Staubli VAL3: AXIS7.pjx

--- AXIS7.pjx ---
Parameters version=s7.2.1 stackSize=5000 millimeterUnit=true
Program file=del.pgx
Program file=find.pgx
Program file=findValue.pgx
Program file=get.pgx
Program file=getSize.pgx
Program file=getType.pgx
Program file=getValue.pgx
Program file=getVelocity.pgx
Program file=loadCycle.pgx
Program file=new.pgx
Program file=onEdit.pgx
Program file=onInsert.pgx
Program file=onProgEnd.pgx
Program file=onRun.pgx
Program file=onStart.pgx
Program file=onStop.pgx
Program file=set.pgx
Program file=setValue.pgx
Program file=setVelocity.pgx
Data file=AXIS7.dtx
Library alias=language path=Disk://kernel/language/language.pjx
Library alias=use path=Disk://kernel/userPage/userPage.pjx

--- AXIS7.dtx ---
public aio MbAI_a8Axispose = {link=ModbusSrv-0\Modbus-Word\MbAI_a8Axispose}
public aio MbAI_aCurPosH = {link=ModbusSrv-0\Modbus-Word\MbAI_aCurPosH}
public aio MbAI_aCurPosL = {link=ModbusSrv-0\Modbus-Word\MbAI_aCurPosL}
public aio MbAI_aUnused4 = {link=ModbusSrv-0\Modbus-Word\MbAI_aUnused4}
public aio MbAI_b8MotorErr = {link=ModbusSrv-0\Modbus-Word\MbAI_b8MotorError}
public aio MbAI_b8MotorPow = {link=ModbusSrv-0\Modbus-Word\MbAI_b8MotorPower}
public aio MbAI_bAxis7Reac = {link=ModbusSrv-0\Modbus-Word\MbAI_bAxis7Reached}
public aio MbAI_bAxis8Reac = {link=ModbusSrv-0\Modbus-Word\MbAI_bAxis8Reached}
public aio MbAI_bBackHome = {link=ModbusSrv-0\Modbus-Word\MbAI_bBackHome}
public aio MbAI_bDownLimit = {link=ModbusSrv-0\Modbus-Word\MbAI_bDownLimit}
public aio MbAI_bEndCycl = {link=ModbusSrv-0\Modbus-Word\MbAI_bEndCycl}
public aio MbAI_bHomeDone = {link=ModbusSrv-0\Modbus-Word\MbAI_bHomeDone}
public aio MbAI_bHomeLimit = {link=ModbusSrv-0\Modbus-Word\MbAI_bHomeLimit}
public aio MbAI_bIsHome = {link=ModbusSrv-0\Modbus-Word\MbAI_bIsHome}
public aio MbAI_bMotorErro = {link=ModbusSrv-0\Modbus-Word\MbAI_bMotorError}
public aio MbAI_bMotorPowe = {link=ModbusSrv-0\Modbus-Word\MbAI_bMotorPower}
public aio MbAI_bOutAlarm = {link=ModbusSrv-0\Modbus-Word\MbAI_bOutAlarm}
public aio MbAI_bPowerOn = {link=ModbusSrv-0\Modbus-Word\MbAI_bPowerOn}
public aio MbAI_bStartCycl = {link=ModbusSrv-0\Modbus-Word\MbAI_bStartCycl}
public aio MbAI_bUnused1 = {link=ModbusSrv-0\Modbus-Word\MbAI_bUnused1}
public aio MbAI_bUnused10 = {link=ModbusSrv-0\Modbus-Word\MbAI_bUnused10}
public aio MbAI_bUnused11 = {link=ModbusSrv-0\Modbus-Word\MbAI_bUnused11}
public aio MbAI_bUnused2 = {link=ModbusSrv-0\Modbus-Word\MbAI_bUnused2}
public aio MbAI_bUnused3 = {link=ModbusSrv-0\Modbus-Word\MbAI_bUnused3}
public aio MbAI_bUnused5 = {link=ModbusSrv-0\Modbus-Word\MbAI_bUnused5}
public aio MbAI_bUnused6 = {link=ModbusSrv-0\Modbus-Word\MbAI_bUnused6}
public aio MbAI_bUnused7 = {link=ModbusSrv-0\Modbus-Word\MbAI_bUnused7}
public aio MbAI_bUnused8 = {link=ModbusSrv-0\Modbus-Word\MbAI_bUnused8}
public aio MbAI_bUnused9 = {link=ModbusSrv-0\Modbus-Word\MbAI_bUnused9}
public aio MbAI_bUpLimit = {link=ModbusSrv-0\Modbus-Word\MbAI_bUpLimit}
public aio MbAO_aAxis7Puls = {link=ModbusSrv-0\Modbus-Word\MbAO_aAxis7Pulse}
public aio MbAO_aAxis8Puls = {link=ModbusSrv-0\Modbus-Word\MbAO_aAxis8Pulse}
public aio MbAO_aJogVelo = {link=ModbusSrv-0\Modbus-Word\MbAO_aJogVelo}
public aio MbAO_aJogVelo8 = {link=ModbusSrv-0\Modbus-Word\MbAO_aJogVelo8}
public aio MbAO_aMoveDis = {link=ModbusSrv-0\Modbus-Word\MbAO_aMoveDis}
public aio MbAO_aMoveDis8 = {link=ModbusSrv-0\Modbus-Word\MbAO_aMoveDis8}
public aio MbAO_aMovePosH = {link=ModbusSrv-0\Modbus-Word\MbAO_aMovePosH}
public aio MbAO_aMovePosH8 = {link=ModbusSrv-0\Modbus-Word\MbAO_aMovePosH8}
public aio MbAO_aMovePosL = {link=ModbusSrv-0\Modbus-Word\MbAO_aMovePosL}
public aio MbAO_aMovePosL8 = {link=ModbusSrv-0\Modbus-Word\MbAO_aMovePosL8}
public aio MbAO_aUnused10 = {link=ModbusSrv-0\Modbus-Word\MbAO_aUnused10}
public aio MbAO_aUnused11 = {link=ModbusSrv-0\Modbus-Word\MbAO_aUnused11}
public aio MbAO_aUnused6 = {link=ModbusSrv-0\Modbus-Word\MbAO_aUnused6}
public aio MbAO_aUnused7 = {link=ModbusSrv-0\Modbus-Word\MbAO_aUnused7}
public aio MbAO_aUnused8 = {link=ModbusSrv-0\Modbus-Word\MbAO_aUnused8}
public aio MbAO_aUnused9 = {link=ModbusSrv-0\Modbus-Word\MbAO_aUnused9}
public aio MbAO_aVelocity = {link=ModbusSrv-0\Modbus-Word\MbAO_aVelocity}
public aio MbAO_aVelocity8 = {link=ModbusSrv-0\Modbus-Word\MbAO_aVelocity8}
public aio MbAO_b7Axis = {link=ModbusSrv-0\Modbus-Word\MbAO_b7Axis}
public aio MbAO_b8Axis = {link=ModbusSrv-0\Modbus-Word\MbAO_b8Axis}
public aio MbAO_bAxis7Dire = {link=ModbusSrv-0\Modbus-Word\MbAO_bAxis7Direction}
public aio MbAO_bAxis7Home = {link=ModbusSrv-0\Modbus-Word\MbAO_bAxis7Home}
public aio MbAO_bAxis8Dire = {link=ModbusSrv-0\Modbus-Word\MbAO_bAxis8Direction}
public aio MbAO_bMoveDir = {link=ModbusSrv-0\Modbus-Word\MbAO_bMoveDir}
public aio MbAO_bMoveDirM = {link=ModbusSrv-0\Modbus-Word\MbAO_bMoveDirM}
public aio MbAO_bMovePos8 = {link=ModbusSrv-0\Modbus-Word\MbAO_bMovePos8}
public aio MbAO_bMoveToPos = {link=ModbusSrv-0\Modbus-Word\MbAO_bMoveToPos}
public aio MbAO_bRecordPos = {link=ModbusSrv-0\Modbus-Word\MbAO_bRecordPos}
public aio MbAO_bResetErr = {link=ModbusSrv-0\Modbus-Word\MbAO_bResetErr}
public aio MbAO_bStopMotor = {link=ModbusSrv-0\Modbus-Word\MbAO_bStopMotor}
public aio MbAO_bUnused1 = {link=ModbusSrv-0\Modbus-Word\MbAO_bUnused1}
public aio MbAO_bUnused2 = {link=ModbusSrv-0\Modbus-Word\MbAO_bUnused2}
public aio MbAO_bUnused3 = {link=ModbusSrv-0\Modbus-Word\MbAO_bUnused3}
public aio MbAO_bUnused4 = {link=ModbusSrv-0\Modbus-Word\MbAO_bUnused4}
public aio MbAO_bUnused5 = {link=ModbusSrv-0\Modbus-Word\MbAO_bUnused5}
public bool bAxisRun
num i = 6
public num nSaveaxis[7]
  [0] = 17569
  [1] = 17753
  [2] = 17775
  [3] = 17555
  [4] = 17803
  [5] = 17805
  [6] = 17722
public num nSaveaxis1[7]
  [0] = 36925
  [1] = 31321
  [2] = 60066
  [3] = 25553
  [4] = 27683
  [5] = 48927
  [6] = 32566
public num nVelocity[7]
  [0] = 8
  [1] = 8
  [2] = 8
  [3] = 8
  [4] = 8
  [5] = 8
  [6] = 8
string l_sItem = "PStart"
public string sItems
public string sSaveaxis[7]
  [0] = "workPos"
  [1] = "p1"
  [2] = "PStart"
  [3] = "P_001"
  [4] = "P_002"
  [5] = "PEnd"
  [6] = "PSychro"

--- del.pgx ---
public program del(num x_nIndex)
begin
  //delete(saveAxis[x_nIndex])
  if size(nSaveaxis)>1
    $ddel(nSaveaxis,x_nIndex)
    $ddel(nSaveaxis1,x_nIndex)
    $ddel(sSaveaxis,x_nIndex)
    $ddel(nVelocity,x_nIndex)
  endIf
end

--- find.pgx ---
public program find(string& x_sItem[], bool& x_bFound[])
begin
  //
  // find one item in the list
  //
  for i=0 to size(sSaveaxis)-1
    if sSaveaxis[i]==x_sItem
      x_bFound=true
      return
    endIf
  endFor
end

--- get.pgx ---
public program get(string& x_sItem[], num x_nIndex)
begin
  //
  // get one element from the list
  //
  x_sItem=sSaveaxis[x_nIndex]
end

--- getSize.pgx ---
public program getSize(num& x_nSize[])
begin
  //
  // get the size of the list
  //
  x_nSize=size(sSaveaxis)
end

--- getValue.pgx ---
public program getValue(num& x_nValue[], num& x_nIndex[], num& x_nValue1[])
begin
  //
  // get the size of the list
  //
  x_nValue=nSaveaxis[x_nIndex]
  //x_nValue=nVelocity[x_nIndex]
  x_nValue1=nSaveaxis1[x_nIndex]
end

--- getVelocity.pgx ---
public program getVelocity(string& x_sItem[], num& x_nVelocity[])
  local num l_nSize
begin
  call getSize(l_nSize)
  for i=0 to l_nSize
    call get(l_sItem,i)
    if l_sItem==x_sItem
      x_nVelocity=nVelocity[i]
      return
      //go back
    endIf
  endFor
end

--- new.pgx ---
public program new(string x_sItem, num x_nIndex)
begin
  // insert a new item
  //insert(saveAxis[x_nIndex])
  $dins(nSaveaxis,size(nSaveaxis))
  $dins(nSaveaxis1,size(nSaveaxis1))
  $dins(sSaveaxis,size(sSaveaxis))
  $dins(nVelocity,size(nVelocity))
  sSaveaxis[size(sSaveaxis)-1]=x_sItem
  nVelocity[size(nVelocity)-1]=8
  ? x_sItem
end

--- onInsert.pgx ---
public program onInsert(string& x_sItem[])
  local string l_sItem
  local string l_sEvent
  local num l_nSize
  local num l_nKey
begin
  //
  // compose the string
  // call getType(l_sItem)
  // x_sItem=l_sItem+" ???"
  //
  // insert all the saveAxis value from the list
  cls()
  call language:message(l_sEvent,65)
  call use:clear(0,13)
  call use:typeCenter(13,l_sEvent,40,true)
  x_sItem=""
  call use:setSizeList(19,0,19,10)
  call use:listcreate("AXIS7")
  l_nSize=size(nSaveaxis)
  for i=0 to l_nSize-1
    l_sEvent=sSaveaxis[i]
    call use:listadd(l_sEvent)
  endFor
  call use:listupdate(0)
  do
    l_nKey=getKey()
    call use:listevent(l_nKey,i,l_sEvent)
    delay(0)
  until l_nKey==255 or l_nKey==270
  if l_nKey==270
    x_sItem="AXIS7>"+l_sEvent
  endIf
  call use:nullKey(l_nKey)
  delay(0)
end

--- onProgEnd.pgx ---
public program onProgEnd(string& x_sItem[])
begin
  //
  // Done, when one program has finished
  //
end

--- onRun.pgx ---
public program onRun(string& x_sItem[])
  local num l_nValue
  local num l_nValue1
  local num l_nVelocity
begin
  //
  // Done, when you execute it
  //
  ////  call findValue(x_sItem,l_nValue)
  ////  aioSet(io:movePulse,l_nValue)
  ////  io:move=true
  ////  delay(0.5)
  ////  io:move=false
  ////  wait(io:atPosition==true or isKeyPressed(255))
  if aioGet(MbAI_bBackHome)!=1
    popUpMsg("7轴未回零位，请先执行回零位操作")
    return
  endIf
  aioSet(MbAO_b7Axis,1)
  aioSet(MbAO_aMoveDis,0)
  aioSet(MbAO_bMoveToPos,0)
  bAxisRun=true
//  aioSet(MbAI_bAxis7Reac,0)
  delay(0.5)
  call findValue(x_sItem,l_nValue,l_nValue1)
  call getVelocity(x_sItem,l_nVelocity)
  l_nVelocity=l_nVelocity*1000/60
  aioSet(MbAO_aMovePosL,l_nValue)
  aioSet(MbAO_aMovePosH,l_nValue1)
  aioSet(MbAO_aVelocity,l_nVelocity)
  aioSet(MbAO_bMoveToPos,1)
  delay(0.5)
  wait(aioGet(MbAI_bAxis7Reac)==0)
  wait(aioGet(MbAI_bAxis7Reac)==1 or isKeyPressed(255))
  if isKeyPressed(255)
    //if !cycleStatus:bCycle and !cycleStatus:bSimulation
      if aioGet(MbAO_bStopMotor)==1
        aioSet(MbAO_bStopMotor,0)
        delay(0.2)
        aioSet(MbAO_bStopMotor,1)
        delay(0.2)
      else
        aioSet(MbAO_bStopMotor,1)
        delay(0.4)
        aioSet(MbAO_bStopMotor,0)
      endIf
    //endIf
  endIf
  aioSet(MbAO_bMoveToPos,0)
  aioSet(MbAO_b7Axis,0)
  logMsg("1")
  // aioSet(io:MbAI_bAxis7Reac,0)
  bAxisRun=false
end

--- onStop.pgx ---
public program onStop(string& x_sItem[])
begin
  //
  // Done after a stop
  //
end

--- set.pgx ---
public program set(string x_sItem, num x_nIndex)
begin
  // set the name
  // saveAxis[x_nIndex].sName=x_sItem
  sSaveaxis[x_nIndex]=x_sItem
end

--- setVelocity.pgx ---
public program setVelocity(num x_nValue, num x_nIndex)
begin
  nVelocity[x_nIndex]=x_nValue
end
